{attribute addProperty BoxType "EP3351-2022-0016"}
{attribute addProperty Id "AIBridge_InputsAT %I*AIBridge_Inputs_EC606E737290AISupply_InputsAT %I*AISupply_Inputs_EC606E737290WcStateAT %I*WcState_F855686C1620InfoDataAT %I*InfoData_BC63D37F80100"}
{attribute addProperty CRC "3250327727"}
{attribute addProperty SizeInBites "240"}
{attribute addProperty SizeInBytes "30"}
TYPE EP3351_606039E3 :
STRUCT
	{attribute addProperty Name "AIBridge_Inputs"}
	AIBridge_Inputs : AIBridge_Inputs_EC606E73;
	{attribute addProperty Name "AISupply_Inputs"}
	AISupply_Inputs : AISupply_Inputs_EC606E73;
	{attribute addProperty Name "WcState"}
	WcState : WcState_F855686C;
	{attribute addProperty Name "InfoData"}
	InfoData : InfoData_BC63D37F;
END_STRUCT
END_TYPE

(* stored: Version 1.2.0.0, ProductVersion 3.1.4024.9
   DUT EP3351_606039E3: Id {187298fe-f11e-4d68-a8ae-56e945447af6} *)
